Universal Robots PolyScope program: 0601.urp

Program 0601 (installation=default directory=/programs/usbdisk/robotics createdIn=5.11.0.108249 lastSavedIn=5.11.0.108249 robotSerialNumber=20215501208)
Calibrated DH parameters: a=[0.000135, -0.201821, -0.391913, -0.000063, 0.000038, 0]; d=[0.162484, -479.507804, 481.562221, -1.92078, 0.099549, 0.099572]; alpha=[1.570789, -0.00078, 0.007148, 1.569147, -1.569841, 0]; deltaTheta=[0, 1.075971, -1.038513, -0.037456, 0, 0]
Robot Program (runOnlyOnce=false)
  Folder init
    Script file /programs/usbdisk/robotics/Init_Variables.script
      | retry_count = 0
      | max_retry = 2
      | fail_flag = 0
      | fail_code = 0
      | current_task = 0
      | 
      | door_state = 0
      | gripper_state = 0
      | dc_motor_state = 0
      | paper_state = 0
    Script file /programs/usbdisk/robotics/Socket_Open.script
      | socket_ok = socket_open("192.168.0.10", 5000)
      | 
      | if socket_ok:
      |   textmsg("Socket open OK")
      |   socket_send_string("PING")
      |   res = socket_read_line()
      |   textmsg("PING response: ", res)
      | else:
      |   textmsg("Socket open FAILED")
      |   halt
      | end
    Call read_door_sensor
SubProgram dc_motor_run (keepSynchronizedWithDisk=false)
  Script file /programs/usbdisk/robotics/DC_Motor_Run.script
    | socket_send_string("D RUN")
    | res = socket_read_line()
    | textmsg("D RUN: ", res)
    | 
    | sleep(2.0)
    | 
    | socket_send_string("D STOP")
    | res = socket_read_line()
    | textmsg("D STOP: ", res)
SubProgram dc_motor_stop (keepSynchronizedWithDisk=false)
  Script file /programs/usbdisk/robotics/DC_Motor_Stop.script
    | socket_send_string("D STOP")
SubProgram gripper_close (keepSynchronizedWithDisk=false)
  Script file /programs/usbdisk/robotics/Gripper_Close.script
    | socket_send_string("G CLOSE")
SubProgram gripper_open (keepSynchronizedWithDisk=false)
  Script file /programs/usbdisk/robotics/Gripper_Open.script
    | socket_send_string("G OPEN")
SubProgram read_camera_result (keepSynchronizedWithDisk=false)
  Script file /programs/usbdisk/robotics/Read_camera_Result.script
    | socket_send_string("V CAMERA")
    | camera_response = socket_read_line()
    | textmsg("Camera: ", camera_response)
SubProgram -> read_door_sensor
SubProgram read_door_sensor (keepSynchronizedWithDisk=false)
  Script file /programs/usbdisk/robotics/Read_Door_Sensor.script
    | socket_send_string("S DOOR")
    | door_response = socket_read_line()
    | textmsg("Door: ", door_response)
